(* CoDeSys 2.3.9.50 project: Steuerung.pro *)
(* Libraries: TcBase.lib 14.5.09 11:14:08, TcSystem.lib 7.6.16 10:01:22, TcBaseMath.lib 27.7.04 11:07:56, TcMath.lib 23.9.04 14:15:30, TcNC.lib 10.10.08 16:55:34, TcMC.lib 27.7.15 07:51:38, TcUtilities.lib 3.2.16 15:08:58, STANDARD.LIB 5.6.98 11:03:02 *)

(* Task configuration *)
TASK Standard (PRIORITY := 0, INTERVAL := T#10ms);
	MAIN
END_TASK

(* Global variable list: Global_Variables *)
VAR_GLOBAL
	(*variables corresponding to the UI elements*)
	start: 					BOOL := FALSE;
	stop: 					BOOL := FALSE;
	pause: 					BOOL := FALSE;
	error: 					BOOL := FALSE;
	quit: 						BOOL := FALSE;
	moveMagazineUp:		BOOL := TRUE;
	bReset: 					BOOL := FALSE;

	(*communication variables for NC axis 1-3*)
	strPLC_TO_NC_Axis_1 AT %Q*:	PlcTONC_AXLESTRUCT;
	strNC_TO_PLC_Axis_1 AT %I*: 	NCTOPLC_AXLESTRUCT;

	strPLC_TO_NC_Axis_2 AT %Q*:	PlcTONC_AXLESTRUCT;
	strNC_TO_PLC_Axis_2 AT %I*: 	NCTOPLC_AXLESTRUCT;

	strPLC_TO_NC_Axis_3 AT %Q*:	PlcTONC_AXLESTRUCT;
	strNC_TO_PLC_Axis_3 AT %I*: 	NCTOPLC_AXLESTRUCT;

	(*outputs to move the pneumatic axis*)
	gripper_on AT %Q*: 			BOOL;
	gripper_down AT %Q*: 			BOOL;
	gripper_up AT%Q*:			BOOL;

	(*inputs of the pneumatic axis*)
	gripper_IsDown AT %I*:		BOOL;
	gripper_IsUp AT %I*:			BOOL;

	(*reference sensors for homing*)
	ref_Axis_2 AT %I*: 				BOOL;
	ref_Axis_3 AT %I*: 				BOOL;

	(*speed modificator. Manipulates how fast each axis moves- must be lower than 1*)
	speedMod: 					LREAL := 1;

	(*emergency stop*)
	stopButton AT %I*:				BOOL;

	(*vacuum sensor*)
	vacuumSensor AT %I*:			BOOL;

	(*UI variables*)
	(*Output - LED*)
	LED_Start AT %Q*: 			BOOL;
	LED_Stop AT %Q*: 			BOOL;
	LED_Quit AT %Q*: 			BOOL;
	LED_Error AT %Q*:			BOOL;

	(*Input - Button*)
	Button_Start AT %I*:			BOOL;
	Button_Stop AT %I*:			BOOL;
	Button_Quit AT %I*:			BOOL;
	Button_Select AT %I*:			BOOL;
	Button_Emergency_1 AT %I*:	BOOL;
	Button_Emergency_2 AT %I*:	BOOL;

	(*emergency stop by the pnoz. true means no emergency*)
	E_Stop AT %I*:				BOOL;
	door_Stop AT %I*:				BOOL;

	(*tray sensors*)
	traySensor_1 AT %I*:			BOOL;
	traySensor_2 AT %I*:			BOOL;




END_VAR

(* Global variable list: persistentVariables *)
VAR_GLOBAL PERSISTENT
	lifetimeCardCounter AT %Q*: 		DWORD		 := 0;
END_VAR

(* Global variable list: Positions *)
VAR_GLOBAL

(*list of positions the axis_2 can reach. need to be tought in*)

	(*first two rows from the reference sensor*)
	Row_1: 		LREAL 		:=	17.0;
	Row_2: 		LREAL 		:= 	82.0;

	(*equals the conveyor belt*)
	Row_3:		LREAL		:= 	243.0;

	(*last two rows form the reference sensor*)
	Row_4: 		LREAL 		:=	403.0;
	Row_5: 		LREAL 		:= 	469.0;

	(*upper most position of the magazine*)
	magazineUp:	LREAL		:= 	-156.0;

END_VAR

(* Global variable list: TwinCAT_Configuration *)
(* Generated automatically by TwinCAT - (read only) *)
VAR_CONFIG
	.strPLC_TO_NC_Axis_1 AT %QB132 : PlcTONC_AXLESTRUCT;	(*  ~ {LinkedWith:TINC^NC-Task 1 SAF^Achsen^Achse 1^Eingänge^Achse 1_FromPlc} *)
	.strNC_TO_PLC_Axis_1 AT %IB136 : NCTOPLC_AXLESTRUCT;	(*  ~ {LinkedWith:TINC^NC-Task 1 SAF^Achsen^Achse 1^Ausgänge^Achse 1_ToPlc} *)
	.strPLC_TO_NC_Axis_2 AT %QB260 : PlcTONC_AXLESTRUCT;	(*  ~ {LinkedWith:TINC^NC-Task 1 SAF^Achsen^Achse 2^Eingänge^Achse 2_FromPlc} *)
	.strNC_TO_PLC_Axis_2 AT %IB264 : NCTOPLC_AXLESTRUCT;	(*  ~ {LinkedWith:TINC^NC-Task 1 SAF^Achsen^Achse 2^Ausgänge^Achse 2_ToPlc} *)
	.strPLC_TO_NC_Axis_3 AT %QB388 : PlcTONC_AXLESTRUCT;	(*  ~ {LinkedWith:TINC^NC-Task 1 SAF^Achsen^Achse 3^Eingänge^Achse 3_FromPlc} *)
	.strNC_TO_PLC_Axis_3 AT %IB392 : NCTOPLC_AXLESTRUCT;	(*  ~ {LinkedWith:TINC^NC-Task 1 SAF^Achsen^Achse 3^Ausgänge^Achse 3_ToPlc} *)
	.gripper_on AT %QX516.0 : BOOL;
	.gripper_down AT %QX516.1 : BOOL;
	.gripper_up AT %QX528.0 : BOOL;
	.gripper_IsDown AT %IX520.0 : BOOL;	(*  ~ {LinkedWith:TIID^Gerät 3 (EtherCAT)^Klemme 6 (CX1100-0004)^Klemme 1 (EL1002)^Channel 1^Input} *)
	.gripper_IsUp AT %IX520.1 : BOOL;	(*  ~ {LinkedWith:TIID^Gerät 3 (EtherCAT)^Klemme 6 (CX1100-0004)^Klemme 1 (EL1002)^Channel 2^Input} *)
	.ref_Axis_2 AT %IX520.2 : BOOL;	(*  ~ {LinkedWith:TIID^Gerät 3 (EtherCAT)^Klemme 6 (CX1100-0004)^Klemme 2 (EL1002)^Channel 2^Input} *)
	.ref_Axis_3 AT %IX520.3 : BOOL;	(*  ~ {LinkedWith:TIID^Gerät 3 (EtherCAT)^Klemme 6 (CX1100-0004)^Klemme 2 (EL1002)^Channel 1^Input} *)
	.stopButton AT %IX524.0 : BOOL;
	.vacuumSensor AT %IX524.1 : BOOL;	(*  ~ {LinkedWith:TIID^Gerät 3 (EtherCAT)^Klemme 6 (CX1100-0004)^Klemme 3 (EL1002)^Channel 1^Input} *)
	.LED_Start AT %QX524.0 : BOOL;	(*  ~ {LinkedWith:TIID^Gerät 3 (EtherCAT)^Klemme 6 (CX1100-0004)^Klemme 14 (EL2008)^Channel 1^Output} *)
	.LED_Stop AT %QX524.1 : BOOL;	(*  ~ {LinkedWith:TIID^Gerät 3 (EtherCAT)^Klemme 6 (CX1100-0004)^Klemme 14 (EL2008)^Channel 3^Output} *)
	.LED_Quit AT %QX524.2 : BOOL;	(*  ~ {LinkedWith:TIID^Gerät 3 (EtherCAT)^Klemme 6 (CX1100-0004)^Klemme 14 (EL2008)^Channel 5^Output} *)
	.LED_Error AT %QX524.3 : BOOL;	(*  ~ {LinkedWith:TIID^Gerät 3 (EtherCAT)^Klemme 6 (CX1100-0004)^Klemme 14 (EL2008)^Channel 7^Output} *)
	.Button_Start AT %IX528.0 : BOOL;	(*  ~ {LinkedWith:TIID^Gerät 3 (EtherCAT)^Klemme 6 (CX1100-0004)^Klemme 4 (EL1004)^Channel 4^Input} *)
	.Button_Stop AT %IX528.1 : BOOL;	(*  ~ {LinkedWith:TIID^Gerät 3 (EtherCAT)^Klemme 6 (CX1100-0004)^Klemme 4 (EL1004)^Channel 3^Input} *)
	.Button_Quit AT %IX528.2 : BOOL;	(*  ~ {LinkedWith:TIID^Gerät 3 (EtherCAT)^Klemme 6 (CX1100-0004)^Klemme 4 (EL1004)^Channel 1^Input} *)
	.Button_Select AT %IX528.3 : BOOL;	(*  ~ {LinkedWith:TIID^Gerät 3 (EtherCAT)^Klemme 6 (CX1100-0004)^Klemme 4 (EL1004)^Channel 2^Input} *)
	.Button_Emergency_1 AT %IX528.4 : BOOL;
	.Button_Emergency_2 AT %IX528.5 : BOOL;
	.E_Stop AT %IX532.0 : BOOL;	(*  ~ {LinkedWith:TIID^Gerät 3 (EtherCAT)^Klemme 6 (CX1100-0004)^Klemme 5 (EL1004)^Channel 1^Input} *)
	.door_Stop AT %IX536.0 : BOOL;
	.traySensor_1 AT %IX532.1 : BOOL;
	.traySensor_2 AT %IX532.2 : BOOL;
	.lifetimeCardCounter AT %QB520 : DWORD;	(*  ~ {LinkedWith:TIID^Gerät 4 (NOV/DP-RAM)^Ausgänge^LifetimeCardCounter} *)
END_VAR

(* POU MAIN, ST *)
PROGRAM MAIN
VAR
	fbFSM :					FSM;
	fbUiWrapper:				UiWrapper;
	cardsPicked:				INT;

(*Testcode*)
	fbPower_Axis_1 : 			MC_Power;
	fbMoveAbsolute_Axis_1 :	MC_MoveAbsolute;
	fbMoveVelocity_Axis_1:	MC_MoveVelocity;
	fbMoveRelative_Axis_1:	MC_MoveRelative;
	fbStop: 					MC_Stop;
	direction :				MC_Direction;
	fbReset_Axis: 			MC_Reset;
	rTrigConvey:				R_TRIG;
	bAxis_Ready: 			BOOL;
	bMove_Absolut_Aborted: 	BOOL;
	bMove_Absolut_Done: 	BOOL;
	bReset_Done: 			BOOL;
	lrAcc_Axis_1: 				LREAL;
	lrActual_Position:			LREAL;
	lrDecel_Axis_1:			LREAL;
	lrJerk_Axis_1: 			LREAL;
	lrPosition_Drive_to:		LREAL;
	lrVelocity_Move_Ab_Axis_1: LREAL;
	lrde: BOOL;
END_VAR
(*ensures speedMod is a valid value*)
speedMod := LIMIT(0, speedMod, 1);

(*cyclic calling of function blocks- "system cycle" *)
fbUiWrapper();
fbFSM();

(*
(*Testcode*)
rTrigConvey(CLK :=roboter_convey_ein);

IF rTrigConvey.Q THEN
	bMoveRelative := TRUE;
END_IF

(*Signal Ventil*)
ventil_ein := roboter_ventil_ein;

(*Freigabesignale werden gesetzt *)
fbPower_Axis_1(
	Enable 			:=	bEnable,
	Enable_Positive 	:= 	bEnable,
	Enable_Negative 	:= 	bEnable,
	Override 			:= 	100.000,
	AxisRefIn 		:= 	strNC_TO_PLC,
	AxisRefOut 		:= 	strPLC_TO_NC,
	status =>,
	Error =>,
	ErrorID =>);

(*Überprüft, ob Achse bereit ist *)
bAxis_Ready := AxisIsReady(strNC_TO_PLC.nStateDWord);

(*Reset der Achse*)
fbReset_Axis(
	Execute			:=	bReset_Axis,
	Axis				:= 	strNC_TO_PLC,
	Done			=>	bReset_Done,
	Error			=>		,
	ErrorID			=>		);

(*Führt eine Absolutbewegung durch*)
fbMoveAbsolute_Axis_1(
	Execute			:=	bMove_Absolut,
	Position			:=	lrPosition_Drive_to,
	Velocity  			:=	lrVelocity_Move_Ab_Axis_1,
	Acceleration		:= 	lrAcc_Axis_1,
	Deceleration		:= 	lrDecel_Axis_1,
	Jerk 			:= 	lrJerk_Axis_1,
	Axis				:= 	strNC_TO_PLC,
	Done			=>	bMove_Absolut_Done,
	CommandAborted=>	bMove_Absolut_Aborted,
	Error			=> 		,
	ErrorID			=>		);

IF fbMoveAbsolute_Axis_1.Done THEN
	bMove_Absolut := FALSE;
END_IF

fbMoveRelative_Axis_1(
    	Execute      		:=	bMoveRelative,
    	Distance     		:=	4000,
    	Velocity     		:=	1500,
	Acceleration		:=	lrAcc_Axis_1,
	Deceleration		:= 	lrDecel_Axis_1,
	Axis				:= 	strNC_TO_PLC,
	Jerk				:=		);

IF fbMoveRelative_Axis_1.Done THEN
	bMoveRelative := FALSE;
END_IF

(*Führt eine Endlosbewegung durch*)
IF bMoveRight THEN
	direction := MC_Positive_Direction;
ELSIF bMoveLeft THEN
	direction := MC_Negative_Direction;
END_IF

fbMoveVelocity_Axis_1(
	Execute			:= 	bMoveRight OR bMoveLeft,
	Velocity			:= 	1500,
	Acceleration		:=	lrAcc_Axis_1,
	Deceleration		:= 	lrDecel_Axis_1,
	Jerk				:= 		,
	Direction			:= 	direction,
	Axis				:= 	strNC_TO_PLC,
	inVelocity		=>		,
	CommandAborted	=>		,
	Error			=>		,
	ErrorId			=>		);

IF bMove_Absolut OR bMoveLeft OR bMoveRight THEN
	bStop := FALSE;
ELSE
	bStop := TRUE;
END_IF

(*Stoppt die Achse*)
fbStop(
	Execute			:=	bStop,
	Deceleration 		:= 	5000,
	Jerk				:=		,
	Axis				:= strNC_TO_PLC,
	Done			=> 		,
	Error			=> 		,
	ErrorID			=> 		);
*)
END_PROGRAM

(* POU FSM, ST *)
FUNCTION_BLOCK FSM
VAR
	state :					INT := 000;
	prevState:				INT := 000;

	errorCounter:				INT := 0;
	rowCounter: 				INT := 0;
	cardCounter:				INT := 0;
	cardsToSort:				INT := 760;

	cardGripped:				BOOL := FALSE;
	safeSorting:				BOOL := FALSE;


	dropTimer :				TON;
	stopTimer:				TON;
	gripperUpImpuls:			TP;
	gripperDownImpuls:		TP;
	doorClosedTrigger:		R_TRIG;

	fbConveyorWrapper:		conveyorWrapper;
	fbMagazineWrapper:		magazineWrapper;
	fbPortalWrapper:			portalWrapper;

END_VAR
fbConveyorWrapper();
fbMagazineWrapper();
fbPortalWrapper();

dropTimer(PT := T#300ms);
stopTimer(IN := Button_Stop, PT := T#1H);
gripperUpImpuls(PT := T#200ms);
gripperDownImpuls(PT := T#200ms);
doorClosedTrigger(CLK := door_Stop);

(*handles the impuls valve of the gripper cylinder*)
gripper_down := gripperDownImpuls.Q;
gripper_up := gripperUpImpuls.Q;

IF NOT error THEN
	bReset := TRUE;
END_IF

(*asynchronous signals*)
(*prevents the second axis from moving while the gripper is down*)
IF gripper_IsDown AND (fbPortalWrapper.bMoveAbsolute OR fbPortalWrapper.bExecuteHome OR fbPortalWrapper.bMoveRelative OR fbPortalWrapper.bMoveLeft OR fbPortalWrapper.bMoveRight) THEN
	dropTimer.IN := FALSE;
	state := 999;
END_IF

(*signal that the conveyor belt has finished its movement*)
IF fbConveyorWrapper.fbMoveRelative.Done THEN
	fbConveyorWrapper.bMoveRelative := FALSE;
END_IF

(*signal that the magazine has finished its movement*)
IF fbMagazineWrapper.fbMoveRelative.Done THEN
	fbMagazineWrapper.bMoveRelative := FALSE;
END_IF

(*checks the vacuum sensor and turns off the ejector*)
IF gripper_on AND NOT vacuumSensor  AND cardGripped THEN
	gripper_on := FALSE;
END_IF

(*emergency stop*)
IF( (NOT E_Stop)  OR (NOT door_Stop)) AND state <> 000 THEN
	dropTimer.IN := FALSE;
	state := 999;
END_IF


(*checks if the trays are properly insertet*)
IF  (traySensor_1 OR traySensor_2) AND state <> 000 THEN
	state := 999;
END_IF

(*pause function. pressing start again continous the process*)
IF MAIN.fbUiWrapper.stopTrigger.Q AND state <> 000  AND state <> 800 THEN
	dropTimer.IN := FALSE;
	prevState := state;
	state := 800;
END_IF

CASE state OF
	(*Init - state*)
	000:
		gripperDownImpuls.IN := FALSE;
		gripperUpImpuls.IN := FALSE;
		stop := TRUE;
		start := FALSE;
		IF MAIN.fbUiWrapper.startTrigger.Q AND (cardCounter < cardsToSort OR Button_Select) THEN
			stop := FALSE;
			pause := FALSE;
			start := TRUE;
			state := 001;
		END_IF

	(*enabling all axis*)
	001:
		fbConveyorWrapper.bEnable := TRUE;
		fbPortalWrapper.bEnable := TRUE;
		fbMagazineWrapper.bEnable:= TRUE;
		gripperUpImpuls.IN := TRUE;
		IF fbConveyorWrapper.bAxis_Ready AND fbPortalWrapper.bAxis_Ready AND fbMagazineWrapper.bAxis_Ready AND gripper_IsUp THEN
			gripperUpImpuls.IN := FALSE;
			state := 002;
		END_IF

	(*checks if the all axis are homed*)
	002:
		IF fbPortalWrapper.bIsHomed  AND fbMagazineWrapper.bIsHomed THEN
			IF Button_Select THEN
				state := 100;
			END_IF
			IF NOT Button_Select  AND strNC_TO_PLC_Axis_3.fPosIst < -5 THEN
				state := 101;
			END_IF
			IF NOT Button_Select AND strNC_TO_PLC_Axis_3.fPosIst > -5 THEN
				state := 999;
			END_IF
		ELSE
			state := 003;
		END_IF

	(*homing state*)
	003:
		fbMagazineWrapper.bExecuteHome := TRUE;
		fbPortalWrapper.bExecuteHome := TRUE;
		IF fbPortalWrapper.bIsHomed  AND fbMagazineWrapper.bIsHomed THEN
			fbPortalWrapper.bExecuteHome := FALSE;
			fbMagazineWrapper.bExecuteHome := FALSE;
			state := 002;
		END_IF

	(*moves magazine in upper position*)
	100:
		fbMagazineWrapper.lrPosition_Drive_to := magazineUp;
		fbMagazineWrapper.bMoveAbsolute := TRUE;
		IF fbMagazineWrapper.fbMoveAbsolute.Done THEN
			(*resets cardCounter when the magazine is moved to the upper pos*)
			cardCounter := 0;
			fbMagazineWrapper.bMoveAbsolute := FALSE;
			state := 101;
		END_IF

	(*move towards and pick up a card*)
	101:
		IF rowCounter > 3 THEN
			rowCounter := 0;
		END_IF
		CASE rowCounter OF
			0:
				fbPortalWrapper.lrPosition_Drive_to := Row_1;
			1:
				fbPortalWrapper.lrPosition_Drive_to := Row_4;
			2:
				fbPortalWrapper.lrPosition_Drive_to := Row_2;
			3:
				fbPortalWrapper.lrPosition_Drive_to := Row_5;
		END_CASE

		fbPortalWrapper.bMoveAbsolute := TRUE;
		IF fbPortalWrapper.fbMoveAbsolute.Done THEN
			fbPortalWrapper.bMoveAbsolute := FALSE;
			state := 102;

			(*counts up for each row picked to select the next target row*)
			rowCounter := rowCounter + 1;
		END_IF

	102:
		gripperDownImpuls.IN := TRUE;
		gripper_on := TRUE;
		IF gripper_IsDown THEN
			gripperDownImpuls.IN := FALSE;
			state := 103;
		END_IF

	103:
		gripper_on := TRUE;
		IF vacuumSensor THEN
			cardGripped := TRUE;
			state := 104;
		END_IF

	104:
		gripperUpImpuls.IN := TRUE;
		IF gripper_IsUp AND vacuumSensor THEN
			gripperUpImpuls.IN := FALSE;
			state := 201;
		END_IF
		IF gripper_IsUp AND NOT  vacuumSensor THEN
			gripperUpImpuls.IN := FALSE;
			errorCounter := errorCounter +1;
			rowCounter := rowCounter - 1;
			rowCounter := LIMIT(0, rowCounter, 3);
			state := 101;
			IF errorCounter > 1 THEN
				error := TRUE;
				state := 997;
			END_IF
		END_IF

	(*move towards conveyor and drop the cards*)
	201:
		fbPortalWrapper.lrPosition_Drive_to := Row_3;
		fbPortalWrapper.bMoveAbsolute := TRUE;
		IF  fbPortalWrapper.fbMoveAbsolute.Done  THEN
			(*card counting for magazine and lifetime*)
			cardCounter := cardCounter + 8;
			lifetimeCardCounter := lifetimeCardCounter + 8;

			fbPortalWrapper.bMoveAbsolute := FALSE;
			IF safeSorting THEN
				state := 202;
			ELSE
				state := 204;
			END_IF
		END_IF
	(*safely dropping the card*)
	202:
		gripper_down := TRUE;
		dropTimer.IN := TRUE;
		IF dropTimer.Q THEN
			dropTimer.IN := FALSE;
			state := 203;
		END_IF

	203:
		gripper_on := FALSE;
		cardGripped := FALSE;
		gripper_down := FALSE;
		IF gripper_IsUp THEN
			state := 205;
		END_IF

	204:
		gripper_on := FALSE;
		cardGripped := FALSE;
		state := 205;

	(*moving state axis 1 and 3*)
	205:
		fbConveyorWrapper.bMoveRelative := TRUE;
		(*starts moving the magazine only after 120 cards to make the magazine larger*)
		IF cardCounter > 120 THEN
			fbMagazineWrapper.bMoveRelative := TRUE;
		END_IF

		IF cardCounter < cardsToSort THEN
			state := 101;
		END_IF
		IF fbConveyorWrapper.fbMoveRelative.Done AND fbMagazineWrapper.fbMoveRelative.Done THEN
			state := 900;
		END_IF

	(*pause state*)
	800:
		fbConveyorWrapper.bStop := TRUE;
		fbPortalWrapper.bStop := TRUE;
		fbMagazineWrapper.bStop := TRUE;
		pause := TRUE;
		bReset := TRUE;
		IF MAIN.fbUiWrapper.startTrigger.Q THEN
			pause := FALSE;
			state := prevState;
		END_IF
		IF stopTimer.ET > T#2S THEN
			fbConveyorWrapper.bMoveRelative := FALSE;
			fbMagazineWrapper.bMoveRelative := FALSE;
			fbMagazineWrapper.bMoveAbsolute := FALSE;
			fbPortalWrapper.bMoveAbsolute := FALSE;
			pause := FALSE;
			state := 997;
		END_IF

	(*end state*)
	900:
		start := FALSE;
		fbConveyorWrapper.bEnable := FALSE;
		fbPortalWrapper.bEnable := FALSE;
		fbMagazineWrapper.bEnable := FALSE;
		state := 000;

	(*error handling. moves gripper and and above the conveyor belt*)
	997:
		bReset := TRUE;
		fbPortalWrapper.bEnable := TRUE;
		gripperUpImpuls.IN := TRUE;
		gripper_on := FALSE;
		cardGripped := FALSE;
		IF gripper_IsUp AND  fbPortalWrapper.bAxis_Ready THEN
			gripperUpImpuls.IN := FALSE;
			IF NOT fbPortalWrapper.bIsHomed  AND NOT fbMagazineWrapper.bIsHomed THEN
				state := 0;
				fbPortalWrapper.bEnable := FALSE;
			ELSE
				state := 998;
			END_IF
		END_IF

	(*error handling. moves gripper and and above the conveyor belt*)
	998:
		fbPortalWrapper.lrPosition_Drive_to := Row_3;
		fbPortalWrapper.bMoveAbsolute := TRUE;
		IF  fbPortalWrapper.fbMoveAbsolute.Done  THEN
			fbPortalWrapper.bMoveAbsolute := FALSE;
			IF error THEN
				state := 999;
			ELSE
				fbConveyorWrapper.bEnable := FALSE;
				fbPortalWrapper.bEnable := FALSE;
				fbMagazineWrapper.bEnable := FALSE;
				state := 000;
			END_IF
		END_IF

	(*error state*)
	999:
		bReset := FALSE;
		error := TRUE;
		start := FALSE;
		fbConveyorWrapper.bEnable := FALSE;
		fbPortalWrapper.bEnable := FALSE;
		fbMagazineWrapper.bEnable := FALSE;

		fbConveyorWrapper.bMoveRelative := FALSE;
		fbMagazineWrapper.bMoveRelative := FALSE;
		fbMagazineWrapper.bMoveAbsolute := FALSE;
		fbPortalWrapper.bMoveAbsolute := FALSE;
		fbPortalWrapper.bExecuteHome := FALSE;
		fbMagazineWrapper.bExecuteHome := FALSE;

		IF MAIN.fbUiWrapper.quitTrigger.Q THEN
			errorCounter := 0;
			bReset := TRUE;
			error := FALSE;
			state := 997;
		END_IF

ELSE
	error := TRUE;
END_CASE;
END_FUNCTION_BLOCK

(* POU conveyorWrapper, ST *)
FUNCTION_BLOCK conveyorWrapper
VAR_INPUT
	lrPosition_Drive_to:			LREAL;
	bExecuteHome:				BOOL;
	bReset_Axis:	 				BOOL;
	bMoveRelative: 				BOOL;
	bMove_Absolut: 				BOOL;
	bStop: 						BOOL;
	bEnable:						BOOL;
	bMoveRight: 					BOOL;
	bMoveLeft: 					BOOL;

END_VAR
VAR_OUTPUT
	bMove_Absolut_Aborted: 		BOOL;
	bMove_Absolut_Done: 		BOOL;
	bReset_Done: 				BOOL;
	bIsHomed: 					BOOL := FALSE;

END_VAR
VAR
	fbPower:		 				MC_Power;
	fbMoveVelocity:				MC_MoveVelocity;
	fbMoveRelative:				MC_MoveRelative;
	fbMoveAbsolute:				MC_MoveAbsolute;
	direction :					MC_Direction;
	fbReset_Axis: 				MC_Reset;
	fbHomeAxis:					MC_Home;
	fbStop: 						MC_Stop;
	fbReset:						MC_Reset;

	bAxis_Ready: 				BOOL;
	maxVelocity: 					LREAL:= 400;
	distance_relative:				LREAL := 900;
END_VAR
(*enables controller *)
fbPower(
	Enable 			:=	bEnable,
	Enable_Positive 	:= 	bEnable,
	Enable_Negative 	:= 	bEnable,
	Override 			:= 	100.000,
	AxisRefIn 		:= 	strNC_TO_PLC_Axis_1,
	AxisRefOut 		:= 	strPLC_TO_NC_Axis_1,
	status 			=>	,
	Error			=>	,
	ErrorID 			=>	);

(*checks if the axis is ready *)
bAxis_Ready := AxisIsReady(strNC_TO_PLC_Axis_1.nStateDWord);

(*reset the axis*)
fbReset_Axis(
	Execute			:=	bReset_Axis,
	Axis				:= 	strNC_TO_PLC_Axis_1,
	Done			=>	bReset_Done,
	Error			=>	,
	ErrorID			=>	);

(*home command of axis*)
fbHomeAxis(
	Execute :=			bExecuteHome,
    	Position  :=			DEFAULT_HOME_POSITION,
   	Axis := 				strNC_TO_PLC_Axis_1,
	AxisOut := 			strPLC_TO_NC_Axis_1);

(*command for realative movement*)
fbMoveRelative(
    	Execute      		:=	bMoveRelative,
    	Distance     		:=	distance_relative,
    	Velocity     		:=	maxVelocity * speedMod,
	Acceleration		:=	,
	Deceleration		:= 	,
	Axis				:= 	strNC_TO_PLC_Axis_1,
	Jerk				:=	);


(*command for endless movement*)
IF bMoveRight THEN
	direction := MC_Positive_Direction;
ELSIF bMoveLeft THEN
	direction := MC_Negative_Direction;
END_IF

fbMoveVelocity(
	Execute			:= 	bMoveRight OR bMoveLeft,
	Velocity			:= 	maxVelocity * speedMod,
	Acceleration		:=	,
	Deceleration		:= 	,
	Jerk				:= 	,
	Direction			:= 	direction,
	Axis				:= 	strNC_TO_PLC_Axis_1,
	inVelocity		=>	,
	CommandAborted	=>	,
	Error			=>	,
	ErrorId			=>	);

IF bMove_Absolut OR bMoveLeft OR bMoveRight THEN
	bStop := FALSE;
ELSE
	bStop := TRUE;
END_IF

(*command for absolute movement*)
fbMoveAbsolute(
	Execute			:=	bMove_Absolut,
	Position			:=	lrPosition_Drive_to,
	Velocity  			:=	maxVelocity * speedMod,
	Acceleration		:= 	,
	Deceleration		:= 	,
	Jerk 			:= 	,
	Axis				:= 	strNC_TO_PLC_Axis_1,
	Done			=>	bMove_Absolut_Done,
	CommandAborted=>	bMove_Absolut_Aborted,
	Error			=> 	,
	ErrorID			=>	);

(*stopps the axis*)
fbStop(
	Execute			:=	bStop,
	Deceleration 		:= 	5000,
	Jerk				:=	,
	Axis				:= 	strNC_TO_PLC_Axis_1,
	Done			=> 	,
	Error			=> 	,
	ErrorID			=> 	);

fbReset(
	Axis				:= 	strNC_TO_PLC_Axis_1,
	Execute 			:= 	bReset);
END_FUNCTION_BLOCK

(* POU magazineWrapper, ST *)
FUNCTION_BLOCK magazineWrapper
VAR_INPUT
	lrPosition_Drive_to:			LREAL;
	bExecuteHome:				BOOL;
	bReset_Axis:	 				BOOL;
	bMoveRelative: 				BOOL;
	bMoveAbsolute: 				BOOL;
	bStop: 						BOOL;
	bEnable:						BOOL;
	bMoveRight: 					BOOL;
	bMoveLeft: 					BOOL;

END_VAR
VAR_OUTPUT
	bMove_Absolut_Aborted: 		BOOL;
	bMove_Absolut_Done: 		BOOL;
	bReset_Done: 				BOOL;
	bIsHomed: 					BOOL := FALSE;

END_VAR
VAR
	fbPower : 					MC_Power;
	fbMoveVelocity:				MC_MoveVelocity;
	fbMoveRelative:				MC_MoveRelative;
	fbMoveAbsolute:				MC_MoveAbsolute;
	direction :					MC_Direction;
	fbReset_Axis: 				MC_Reset;
	fbHomeAxis:					MC_Home;
	fbStop: 						MC_Stop;
	fbReset:						MC_Reset;
	bAxis_Ready: 				BOOL;
	maxVelocity: 					LREAL:= 3;
	distance_relative:				LREAL := 1.95;
END_VAR
(*enables controller *)
fbPower(
	Enable 			:=	bEnable,
	Enable_Positive 	:= 	bEnable,
	Enable_Negative 	:= 	bEnable,
	Override 			:= 	100.000,
	AxisRefIn 		:= 	strNC_TO_PLC_Axis_3,
	AxisRefOut 		:= 	strPLC_TO_NC_Axis_3,
	status 			=>	,
	Error			=>	,
	ErrorID 			=>	);

(*checks if the axis is ready *)
bAxis_Ready := AxisIsReady(strNC_TO_PLC_Axis_3.nStateDWord);

(*reset the axis*)
fbReset_Axis(
	Execute			:=	bReset_Axis,
	Axis				:= 	strNC_TO_PLC_Axis_3,
	Done			=>	bReset_Done,
	Error			=>	,
	ErrorID			=>	);

(*home command of axis*)
fbHomeAxis(
	Execute :=			bExecuteHome,
    	Position  :=			DEFAULT_HOME_POSITION,
	bCalibrationCam := 	ref_Axis_3,
   	Axis := 				strNC_TO_PLC_Axis_3,
	AxisOut := 			strPLC_TO_NC_Axis_3);

IF fbHomeAxis.Done THEN
	bIsHomed := TRUE;
END_IF

(*command for realative movement*)
fbMoveRelative(
    	Execute      		:=	bMoveRelative,
    	Distance     		:=	distance_relative,
    	Velocity     		:=	maxVelocity * speedMod,
	Acceleration		:=	,
	Deceleration		:= 	,
	Axis				:= 	strNC_TO_PLC_Axis_3,
	Jerk				:=	);


(*command for endless movement*)
IF bMoveRight THEN
	direction := MC_Positive_Direction;
ELSIF bMoveLeft THEN
	direction := MC_Negative_Direction;
END_IF

fbMoveVelocity(
	Execute			:= 	bMoveRight OR bMoveLeft,
	Velocity			:= 	maxVelocity * speedMod,
	Acceleration		:=	,
	Deceleration		:= 	,
	Jerk				:= 	,
	Direction			:= 	direction,
	Axis				:= 	strNC_TO_PLC_Axis_3,
	inVelocity		=>	,
	CommandAborted	=>	,
	Error			=>	,
	ErrorId			=>	);

IF bMoveAbsolute OR bMoveLeft OR bMoveRight THEN
	bStop := FALSE;
ELSE
	bStop := TRUE;
END_IF

(*command for absolute movement*)
fbMoveAbsolute(
	Execute			:=	bMoveAbsolute,
	Position			:=	lrPosition_Drive_to,
	Velocity  			:=	6,
	Acceleration		:= 	,
	Deceleration		:= 	,
	Jerk 			:= 	,
	Axis				:= 	strNC_TO_PLC_Axis_3,
	Done			=>	bMove_Absolut_Done,
	CommandAborted=>	bMove_Absolut_Aborted,
	Error			=> 	,
	ErrorID			=>	);

(*stopps the axis*)
fbStop(
	Execute			:=	bStop,
	Deceleration 		:= 	5000,
	Jerk				:=	,
	Axis				:= 	strNC_TO_PLC_Axis_3,
	Done			=> 	,
	Error			=> 	,
	ErrorID			=> 	);

fbReset(
	Axis				:= 	strNC_TO_PLC_Axis_3,
	Execute 			:= 	bReset);
END_FUNCTION_BLOCK

(* POU portalWrapper, ST *)
FUNCTION_BLOCK portalWrapper
VAR_INPUT
	lrPosition_Drive_to:			LREAL;
	bExecuteHome:				BOOL;
	bReset_Axis:	 				BOOL;
	bMoveRelative: 				BOOL;
	bMoveAbsolute: 				BOOL;
	bStop: 						BOOL;
	bEnable:						BOOL;
	bMoveRight: 					BOOL;
	bMoveLeft: 					BOOL;
	bMove_Absolut: 				BOOL;

END_VAR
VAR_OUTPUT
	bMove_Absolut_Aborted: 		BOOL;
	bMove_Absolut_Done: 		BOOL;
	bReset_Done: 				BOOL;
	bIsHomed: 					BOOL := FALSE;

END_VAR
VAR
	fbPower : 					MC_Power;
	fbMoveVelocity:				MC_MoveVelocity;
	fbMoveRelative:				MC_MoveRelative;
	fbMoveAbsolute:				MC_MoveAbsolute;
	direction :					MC_Direction;
	fbReset_Axis: 				MC_Reset;
	fbHomeAxis:					MC_Home;
	fbStop: 						MC_Stop;
	fbReset:						MC_Reset;
	bAxis_Ready: 				BOOL;
	maxVelocity: 					LREAL:= 550;
	distance_relative:				LREAL := 200;
END_VAR
(*enables controller *)
fbPower(
	Enable 			:=	bEnable,
	Enable_Positive 	:= 	bEnable,
	Enable_Negative 	:= 	bEnable,
	Override 			:= 	100.000,
	AxisRefIn 		:= 	strNC_TO_PLC_Axis_2,
	AxisRefOut 		:= 	strPLC_TO_NC_Axis_2,
	status 			=>	,
	Error			=>	,
	ErrorID 			=>	);

(*checks if the axis is ready *)
bAxis_Ready := AxisIsReady(strNC_TO_PLC_Axis_2.nStateDWord);

(*reset the axis*)
fbReset_Axis(
	Execute			:=	bReset_Axis,
	Axis				:= 	strNC_TO_PLC_Axis_2,
	Done			=>	bReset_Done,
	Error			=>	,
	ErrorID			=>	);

(*home command of axis*)
fbHomeAxis(
	Execute :=			bExecuteHome,
    	Position  :=			DEFAULT_HOME_POSITION,
	bCalibrationCam := 	ref_Axis_2,
   	Axis := 				strNC_TO_PLC_Axis_2,
	AxisOut := 			strPLC_TO_NC_Axis_2);

IF fbHomeAxis.Done THEN
	bIsHomed := TRUE;
END_IF


(*command for realative movement*)
fbMoveRelative(
    	Execute      		:=	bMoveRelative,
    	Distance     		:=	distance_relative,
    	Velocity     		:=	maxVelocity * speedMod,
	Acceleration		:=	,
	Deceleration		:= 	,
	Axis				:= 	strNC_TO_PLC_Axis_2,
	Jerk				:=	);


(*command for endless movement*)
IF bMoveRight THEN
	direction := MC_Positive_Direction;
ELSIF bMoveLeft THEN
	direction := MC_Negative_Direction;
END_IF

fbMoveVelocity(
	Execute			:= 	bMoveRight OR bMoveLeft,
	Velocity			:= 	maxVelocity * speedMod,
	Acceleration		:=	,
	Deceleration		:= 	,
	Jerk				:= 	,
	Direction			:= 	direction,
	Axis				:= 	strNC_TO_PLC_Axis_2,
	inVelocity		=>	,
	CommandAborted	=>	,
	Error			=>	,
	ErrorId			=>	);

IF bMoveAbsolute OR bMoveLeft OR bMoveRight THEN
	bStop := FALSE;
ELSE
	bStop := TRUE;
END_IF

(*command for absolute movement*)
fbMoveAbsolute(
	Execute			:=	bMoveAbsolute,
	Position			:=	lrPosition_Drive_to,
	Velocity  			:=	maxVelocity * speedMod,
	Acceleration		:= 	,
	Deceleration		:= 	,
	Jerk 			:= 	,
	Axis				:= 	strNC_TO_PLC_Axis_2,
	Done			=>	bMove_Absolut_Done,
	CommandAborted=>	bMove_Absolut_Aborted,
	Error			=> 	,
	ErrorID			=>	);


(*stopps the axis*)
fbStop(
	Execute			:=	bStop,
	Deceleration 		:= 	5000,
	Jerk				:=	,
	Axis				:= 	strNC_TO_PLC_Axis_2,
	Done			=> 	,
	Error			=> 	,
	ErrorID			=> 	);

fbReset(
	Axis				:= 	strNC_TO_PLC_Axis_2,
	Execute 			:= 	bReset);
END_FUNCTION_BLOCK

(* POU UiWrapper, ST *)
FUNCTION_BLOCK UiWrapper
VAR_INPUT
END_VAR
VAR_OUTPUT
END_VAR
VAR
	startTrigger: 				R_TRIG;
	stopTrigger: 				R_TRIG;
	quitTrigger: 				R_TRIG;
	moveMagazineUpTrigger: 	R_TRIG;

	blinkTimer:				TON;
END_VAR
(*trigger to check for button presses*)
startTrigger(CLK := Button_Start);
quitTrigger(CLK := Button_Quit);
moveMagazineUpTrigger(CLK := Button_Select);
stopTrigger(CLK := Button_Stop);

(*connects plc variables to buttons and leds*)
LED_Error := error;
LED_Start := start;
LED_Stop := stop OR pause;

IF error THEN
	blinkTimer(IN := NOT blinkTimer.Q, PT := T#1.5S);

END_IF
IF blinkTimer.Q THEN
	LED_Quit := NOT LED_Quit;
END_IF
IF quitTrigger.Q THEN
	LED_Quit := FALSE;
END_IF
END_FUNCTION_BLOCK

(* Visualisation UI
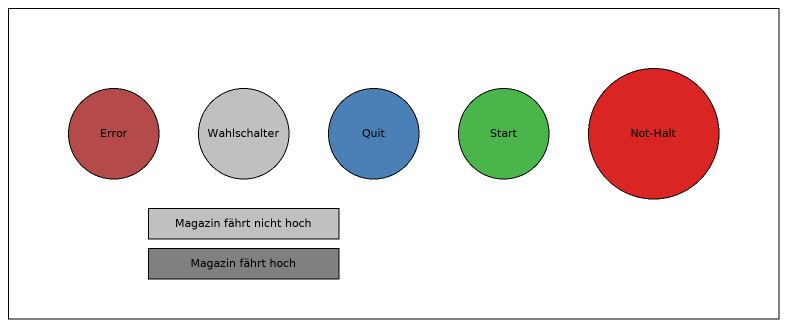
ellipse at (70,90)-(161,181): text "Error"; alarm colour if error
ellipse at (200,90)-(291,181): text "Wahlschalter"; alarm colour if moveMagazineUp; toggles moveMagazineUp
ellipse at (330,90)-(421,181): text "Quit"; alarm colour if quit; toggles quit
ellipse at (590,70)-(721,201): text "Not-Halt"
ellipse at (460,90)-(551,181): text "Start"; alarm colour if start; toggles start
rectangle at (150,210)-(341,241): text "Magazin fährt nicht hoch"
rectangle at (150,250)-(341,281): text "Magazin fährt hoch"
1 more shapes without text or variables
*)
